INTERFACE ITF_MessengerSender

METHOD SendData_BOOL : BOOL
VAR_INPUT
	sNazwa		: STRING;
	itfNadawca	: ITF_MessengerSender;
END_VAR
END_METHOD

METHOD SendData_REAL : BOOL
VAR_INPUT
	sNazwa		: STRING;
	rWartosc	: REAL;
	itfNadawca	: ITF_MessengerSender;
END_VAR
END_METHOD

END_INTERFACE

(* stored: Version 1.1.0.1
   Itf ITF_MessengerSender: Id {f2c748b8-07c6-03cf-04c2-0bcc78ff32eb}
   Method SendData_BOOL: Id {298a0d8a-859a-0345-1b64-39c0a67da553}
   Method SendData_REAL: Id {90c1e12c-5b0c-0772-240d-9c9ad6717b88} *)
